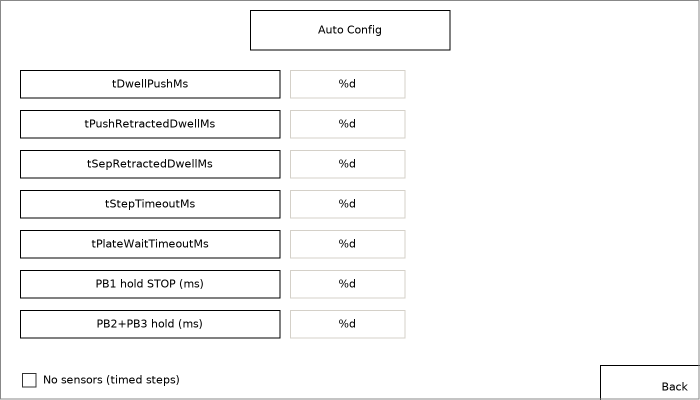
VISUALIZATION AutoConfig  // 700x400
VAR_IN_OUT
	stMasterAutoCycle : ST_HmiMasterAuto;
	stCfg : ST_HmiMasterAutoCfg;
END_VAR
    Rectangle (250,10 200x40), "Auto Config"
    Checkbox (20,365 240x30), "No sensors (timed steps)", variable: GVL_HmiPersistent.stMasterAutoCfg.bNoSensors
    Checkbox (20,405 240x30), "Bypass plate sensors", variable: GVL_HmiPersistent.stMasterAutoCfg.bBypassPlateSensors
    Rectangle (20,70 260x28), "tDwellPushMs"
    Textfield (290,70 115x28), "%d", text variable: GVL_HmiPersistent.stMasterAutoCfg.tDwellPushMs
        OnMouseClick: write the text variable via Default
    Rectangle (20,110 260x28), "tPushRetractedDwellMs"
    Textfield (290,110 115x28), "%d", text variable: GVL_HmiPersistent.stMasterAutoCfg.tPushRetractedDwellMs
        OnMouseClick: write the text variable via Default
    Rectangle (20,150 260x28), "tSepRetractedDwellMs"
    Textfield (290,150 115x28), "%d", text variable: GVL_HmiPersistent.stMasterAutoCfg.tSepRetractedDwellMs
        OnMouseClick: write the text variable via Default
    Rectangle (20,190 260x28), "tStepTimeoutMs"
    Textfield (290,190 115x28), "%d", text variable: GVL_HmiPersistent.stMasterAutoCfg.tStepTimeoutMs
        OnMouseClick: write the text variable via Default
    Rectangle (20,230 260x28), "tPlateWaitTimeoutMs"
    Textfield (290,230 115x28), "%d", text variable: GVL_HmiPersistent.stMasterAutoCfg.tPlateWaitTimeoutMs
        OnMouseClick: write the text variable via Default
    Rectangle (20,270 260x28), "PB1 hold STOP (ms)"
    Textfield (290,270 115x28), "%d", text variable: GVL_HmiPersistent.stMasterAutoCfg.tPbStopHoldMs
        OnMouseClick: write the text variable via Default
    Rectangle (20,310 260x28), "PB2+PB3 hold (ms)"
    Textfield (290,310 115x28), "%d", text variable: GVL_HmiPersistent.stMasterAutoCfg.tPbStartHoldMs
        OnMouseClick: write the text variable via Default
    Rectangle (600,365 150x44), "Back"
        OnMouseDown: change screen: Main
END_VISUALIZATION

(* stored: Version 1.1.0.1, ProductVersion 3.1.4024.16
   Visu AutoConfig: Id {bd141093-4f61-5aab-ad0e-82f19e6b8457} *)
